// TIA Portal V17 program export: 1 tag tables, 0 data types, 0 data blocks, 3 code blocks (in call order from the OBs), 0 instance data blocks

VAR_GLOBAL   // PLC tag table "Default tag table"
   "high sensor" AT %I0.0 : Bool;
   "low sensor" AT %I0.1 : Bool;
   "pallet sensor" AT %I0.2 : Bool;
   "loaded sensor" AT %I0.3 : Bool;
   "at the left entry" AT %I0.4 : Bool;
   "at the left exit" AT %I0.5 : Bool;
   "at right entry" AT %I0.6 : Bool;
   "at right exit" AT %I0.7 : Bool;
   start AT %I1.0 : Bool;
   reset AT %I1.1 : Bool;
   stop AT %I1.2 : Bool;
   "Emergency stop" AT %I1.3 : Bool;
   auto AT %I1.4 : Bool;
   "factory runnning" AT %I1.5 : Bool;
   "conveyor enter" AT %Q0.0 : Bool;
   load AT %Q0.1 : Bool;
   unload AT %Q0.2 : Bool;
   "transfer left" AT %Q0.3 : Bool;
   "transfer right" AT %Q0.4 : Bool;
   "conveyor left" AT %Q0.5 : Bool;
   "conveyor right" AT %Q0.6 : Bool;
   "start light" AT %Q0.7 : Bool;
   "Reset light" AT %Q1.0 : Bool;
   "stop light" AT %Q1.1 : Bool;
   "counter" AT %QW30 : Int;
END_VAR

ORGANIZATION_BLOCK "Main"   // OB1, LAD, ProgramCycle
TITLE = "Main Program Sweep (Cycle)"
VERSION : 0.1
// stored: IsIECCheckEnabled false
   VAR_TEMP
      OB1_EV_CLASS : Byte;   // Bits 0-3 = 1 (Coming event), Bits 4-7 = 1 (Event class 1)
      OB1_SCAN_1 : Byte;   // 1 (Cold restart scan 1 of OB 1), 3 (Scan 2-n of OB 1)
      OB1_PRIORITY : Byte;   // Priority of OB Execution
      OB1_OB_NUMBR : Byte;   // 1 (Organization block 1, OB1)
      OB1_RESERVED_1 : Byte;   // Reserved for system
      OB1_RESERVED_2 : Byte;   // Reserved for system
      OB1_PREV_CYCLE : Int;   // Cycle time of previous OB1 scan (milliseconds)
      OB1_MIN_CYCLE : Int;   // Minimum cycle time of OB1 (milliseconds)
      OB1_MAX_CYCLE : Int;   // Maximum cycle time of OB1 (milliseconds)
      OB1_DATE_TIME : Date_And_Time;   // Date and time OB1 started
   END_VAR
BEGIN

REGION Network 1
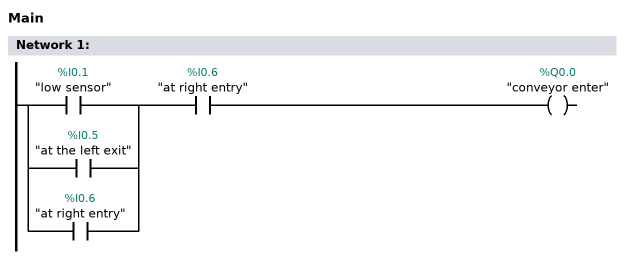
   RUNG wire#powerrail
      Contact( "low sensor" )
      wire#w1
      Contact( "at right entry" )
      Coil( "conveyor enter" )
   END_RUNG
   RUNG wire#powerrail
      Contact( "at the left exit" )
   END_RUNG wire#w1
   RUNG wire#powerrail
      Contact( "at right entry" )
   END_RUNG wire#w1
   // the same network as SCL:
   "conveyor enter" := ("low sensor" OR "at the left exit" OR "at right entry") AND "at right entry";
END_REGION
END_ORGANIZATION_BLOCK

FUNCTION "FC_1" : Void   // FC1, LAD
VERSION : 0.1
// stored: AutoNumber true, IsIECCheckEnabled false, UDAEnableTagReadback false
BEGIN

REGION Network 1
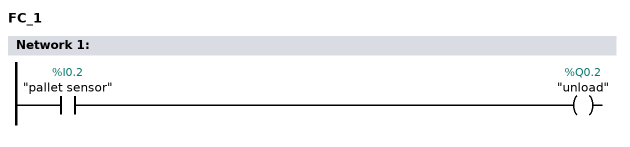
   RUNG wire#powerrail
      Contact( "pallet sensor" )
      Coil( "unload" )
   END_RUNG
   // the same network as SCL:
   "unload" := "pallet sensor";
END_REGION
END_FUNCTION

FUNCTION "FC_2" : Void   // FC2, LAD
VERSION : 0.1
// stored: AutoNumber true, IsIECCheckEnabled false, UDAEnableTagReadback false
BEGIN
END_FUNCTION
